# EPICS substitutions: sdgApp/Db/sdg-3.substitutions
file sdg01.template
{
pattern{ N, S }
       { 1, A }
       { 2, B }
       { 3, C }
}
